FUNCTION_BLOCK L3_Cinta EXTENDS L1_ModuleBase

VAR_INPUT
	Situar: BOOL;
	Transferir: BOOL;
END_VAR

VAR_OUTPUT
	fbController	: L2_Cinta_SFC:=(dr:=dr);
	pp				: L1_Sensor;
	cp0				: L1_Sensor;
	cp1				: L1_Sensor;
	cp2				: L1_Sensor;
	RUN				: L1_Actuator;
	REV				: L1_Actuator;
	R_1				: L1_Actuator;
	S_1				: L1_Actuator;

	// colores para distingur cuándo situa y cuándo transfiere	
	colPicFramTransferir : DWORD;
	colPicFillTransferir : DWORD;

	colPicFramSituar : DWORD;
	colPicFillSituar : DWORD;
	
END_VAR

METHOD Avanza : BOOL
VAR_INPUT
END_VAR
RUN.ForceValue(NewValue := TRUE);
REV.ForceValue(NewValue := FALSE);
END_METHOD

METHOD ProcessCycle : BOOL 
VAR_INPUT
	dr			: REFERENCE TO L1_Director;
	tapas		: REFERENCE TO L6_Tapas;	
END_VAR
// Sensores y condiciones iniciales
pp.ProcessCycle(LocalHost:=dr.gmLocalHost, sfcValue=>fbController.pp);
cp0.ProcessCycle(LocalHost:=dr.gmLocalHost, sfcValue=>fbController.cp0);
cp1.ProcessCycle(LocalHost:=dr.gmLocalHost, sfcValue=>fbController.cp1);
cp2.ProcessCycle(LocalHost:=dr.gmLocalHost, sfcValue=>fbController.cp2);
IC := TRUE;

// Actuadores y actualización de tapas
fbController.ProcessCycle(dr.gmModeActual);
fbController(Situar := Situar, Transferir := Transferir,	
	dr:=dr, IC:=IC, Execute:=Execute, Ack:=Ack, Ready=>Ready, Done=>Done);

RUN.ProcessCycle(gmMode:=dr.gmModeActual, sfcValue:=fbController.RUN);
REV.ProcessCycle(gmMode:=dr.gmModeActual, sfcValue:=fbController.REV);
R_1.ProcessCycle(gmMode:=dr.gmModeActual, sfcValue:=fbController.R_1);
S_1.ProcessCycle(gmMode:=dr.gmModeActual, sfcValue:=fbController.S_1);

// Actualizar las flechas de la cinta dependiendo de si sitúa o transfiere
colPicFramTransferir := SEL(Transferir, colModFramReady, fbController.colPicFram);
colPicFillTransferir := SEL(Transferir, colModFillReady, fbController.colPicFill);
colPicFramSituar	 := SEL(Situar, 	colModFramReady, fbController.colPicFram);
colPicFillSituar	 := SEL(Situar, 	colModFillReady, fbController.colPicFill);
END_METHOD

METHOD Retrocede : BOOL
VAR_INPUT
END_VAR
RUN.ForceValue(NewValue := TRUE);
REV.ForceValue(NewValue := TRUE);
END_METHOD

END_FUNCTION_BLOCK

(* stored: Version 1.1.0.1, ProductVersion 3.1.4024.11
   POU L3_Cinta: Id {f4de692b-96c6-493e-9b33-3a90e20acfad}, SpecialFunc None
   Method Avanza: Id {962ac213-4605-4eb0-b4f2-71abfc5eecac}
   Method ProcessCycle: Id {8ef223d1-a933-4fe3-87e8-40d9ed750433}
   Method Retrocede: Id {319ef3db-3f91-40fc-bb86-4c3e886a06cc} *)
